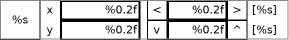
VISUALIZATION _VISU_PlacementXY  // 289x40
VAR_IN_OUT
	m_Inst : FB_PointCorr;  
END_VAR
    Rectangle (40,0 20x20), "x"
    Rectangle (40,20 20x20), "y"
    Rectangle (0,0 40x40), "%s", text variable: m_Inst._aName
    Rectangle (249,20 40x20), "[%s]", text variable: m_Inst._aUnit
    Rectangle (249,0 40x20), "[%s]", text variable: m_Inst._aUnit
    Rectangle (60,0 80x20), "%0.2f", tooltip "reference", text variable: m_Inst._fX_Ref
        OnMouseClick: write the text variable via Default
    Rectangle (60,20 80x20), "%0.2f", tooltip "reference", text variable: m_Inst._fY_Ref
        OnMouseClick: write the text variable via Default
    RoundedRectangle (147,0 20x20), "<"
        p3092690914: m_Inst.nBtnColor
        p2167032090: m_Inst.nBtnColor
        tap m_Inst.bCmd_X_plus
    RoundedRectangle (227,0 20x20), ">"
        p3092690914: m_Inst.nBtnColor
        p2167032090: m_Inst.nBtnColor
        tap m_Inst.bCmd_X_minus
    RoundedRectangle (147,20 20x20), "v"
        p3092690914: m_Inst.nBtnColor
        p2167032090: m_Inst.nBtnColor
        tap m_Inst.bCmd_Y_plus
    RoundedRectangle (227,20 20x20), "^"
        p3092690914: m_Inst.nBtnColor
        p2167032090: m_Inst.nBtnColor
        tap m_Inst.bCmd_Y_minus
    Rectangle (167,0 60x20), "%0.2f", tooltip "correction relative", text variable: m_Inst._fX_Pos
        OnMouseClick: write the text variable via Default
    Rectangle (167,20 60x20), "%0.2f", tooltip "correction relative", text variable: m_Inst._fY_Pos
        OnMouseClick: write the text variable via Default
END_VISUALIZATION

(* stored: Version 1.1.0.1, ProductVersion 3.1.4024.3
   Visu _VISU_PlacementXY: Id {17f498b7-d2c9-4c22-ab4b-3f8a77be311b} *)
